FUNCTION_BLOCK FB_UpdateIO
VAR_INPUT
END_VAR
VAR_OUTPUT
END_VAR
VAR
END_VAR

END_FUNCTION_BLOCK

(* stored: Version 1.1.0.1, ProductVersion 3.1.4024.0
   POU FB_UpdateIO: Id {02be4b73-c84a-06dc-2810-905d0b106449}, SpecialFunc None *)
